// TIA Portal V17 export
// export: Created 2022-07-20T07:02:37.9315694Z, ExportSetting WithDefaults, DisplayName Totally Integrated Automation Portal, DisplayVersion V17, DisplayName TIA Portal Openness, DisplayVersion V17, DisplayName TIA Portal Version Control Interface, DisplayVersion V17, DisplayName SINAMICS Startdrive Advanced, DisplayVersion V17, DisplayName SINAMICS Startdrive G130, G150, S120, S150, SINAMICS MV, S210, DisplayVersion V17, DisplayName SINAMICS Startdrive G110M, G120, G120C, G120D, G120P, G115D, DisplayVersion V17, DisplayName STEP 7 Professional, DisplayVersion V17, DisplayName STEP 7 Safety, DisplayVersion V17, DisplayName WinCC Advanced, DisplayVersion V17
VAR_GLOBAL   // PLC tag table "UltrasonicSensor_Baumer_CommunicationTable"
   Baumer_Unwinder_Input_Specifics AT %IB188 : Byte;
   Baumer_Unwinder_Input_Scale AT %IB192 : SInt;
   Baumer_1_Output_ProcessData AT %QB474 : Byte;
   Baumer_Unwinder_Input_Value AT %ID188 : DWord;
   Baumer_RewinderBottom_Input_Specifics AT %IB798 : Byte;
   Baumer_RewinderBottom_Input_Scale AT %IB802 : SInt;
   Baumer_RewinderBottom_Input_Value AT %ID798 : DWord;
END_VAR
